Universal Robots PolyScope program: _adminCG-InvBToPHome.urp

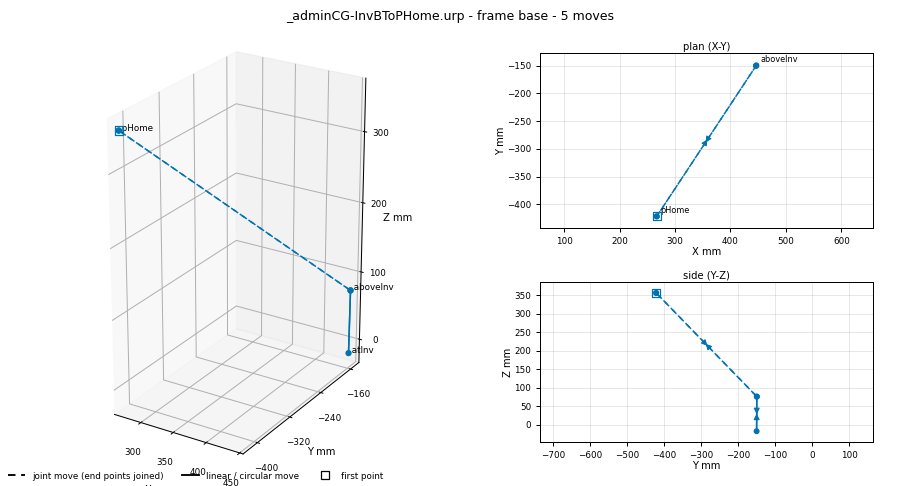
[picture p0: tool path of _adminCG-InvBToPHome.urp in frame base, 5 of 5 moves have a stored position in this frame; points joined in program order, loops and branches not executed]
Program _adminCG-InvBToPHome (installation=admin directory=/programs/THU_530PM createdIn=3.8.0.61336 lastSavedIn=3.15.8.106339 robotSerialNumber=2015350924)
Calibrated DH parameters: a=[0, -0.425, -0.39225, 0, 0, 0]; d=[0.089159, 0, 0, 0.10915, 0.09465, 0.0823]; alpha=[1.570796, 0, 0, 1.570796, -1.570796, 0]; deltaTheta=[0, 0, 0, 0, 0, 0]
Robot Program (runOnlyOnce=true)
  Set DigitalOutput pin=digital_out[0]; digitalValue=0
  Call _adminLinearIndex2
  MoveJ speed 60 deg/s, acceleration 80 deg/s^2 (useActiveTCP=true)
    Waypoint pHome: TCP in base x=267.077 y=-421.526 z=355.862 mm, rx=1.114 ry=1.1061 rz=0.0051 rad; joints [-45.007, -90.005, -89.993, -90.005, 90, -0.004] deg; flange x=267.08 y=-421.53 z=431.862 mm, rx=1.2021 ry=-2.9025 rz=-0.0001 rad
    Waypoint aboveInv: TCP in base x=446.522 y=-149.612 z=75.742 mm, rx=1.1163 ry=1.1067 rz=-0.0014 rad; joints [-5.099, -101.028, -122.856, -46.337, 89.934, 40.185] deg; flange x=446.821 y=-149.55 z=151.741 mm, rx=1.1935 ry=-2.9018 rz=-0.0012 rad
  MoveL speed 250 mm/s, acceleration 1200 mm/s^2 (useActiveTCP=true) feature=Base
    Waypoint atInv: TCP in base x=445.929 y=-150.177 z=-17.742 mm, rx=1.1163 ry=1.1068 rz=-0.0015 rad; joints [-5.175, -113.085, -126.768, -30.375, 89.929, 40.11] deg; flange x=446.238 y=-150.111 z=58.258 mm, rx=1.1935 ry=-2.9016 rz=-0.0012 rad
    Set DigitalOutput pin=digital_out[0]; digitalValue=1
    Wait Sleep waitTime=1
    Waypoint aboveInv: TCP in base x=446.522 y=-149.612 z=75.742 mm, rx=1.1163 ry=1.1067 rz=-0.0014 rad; joints [-5.099, -101.028, -122.856, -46.337, 89.934, 40.185] deg; flange x=446.821 y=-149.55 z=151.741 mm, rx=1.1935 ry=-2.9018 rz=-0.0012 rad
  MoveJ speed 180 deg/s, acceleration 100 deg/s^2 (useActiveTCP=true)
    Waypoint pHome: TCP in base x=267.077 y=-421.526 z=355.862 mm, rx=1.114 ry=1.1061 rz=0.0051 rad; joints [-45.007, -90.005, -89.993, -90.005, 90, -0.004] deg; flange x=267.08 y=-421.53 z=431.862 mm, rx=1.2021 ry=-2.9025 rz=-0.0001 rad
SubProgram  [hidden by the author, left out]
SubProgram _adminLinearIndex2 [hidden by the author, left out]
